TYPE XtsHardwareInfo :
STRUCT
	NoOfParts: UDINT;
	NoOfTracks : UDINT;
	NoOfModules : ARRAY[1..10] OF UDINT;
	HWState : XtsHardwareState;
END_STRUCT
END_TYPE

(* stored: Version 1.1.0.1, ProductVersion 3.1.4024.11
   DUT XtsHardwareInfo: Id {304f91e0-1afd-4f2f-84e9-27faf5187ca4} *)
